// TIA Portal V17 export
// export: Created 2025-03-05T08:03:47.5129937Z, ExportSetting WithDefaults, DisplayName Totally Integrated Automation Portal, DisplayVersion V17 Update 8, DisplayName TIA Portal Openness, DisplayVersion V17 Update 8, DisplayName TIA Portal Version Control Interface, DisplayVersion V17, DisplayName SINAMICS Startdrive Advanced, DisplayVersion V17 SP2, DisplayName SINAMICS Startdrive G110M, G120, G120C, G120D, G120P, G115D, DisplayVersion V17 SP2, DisplayName SINAMICS Startdrive G130, G150, S120, S150, SINAMICS MV, S210, DisplayVersion V17 SP2, DisplayName STEP 7 Professional, DisplayVersion V17 Update 8, DisplayName SINUMERIK ONE STEP 7 Toolbox, DisplayVersion V17 Update 12, DisplayName SINUMERIK 840D sl STEP 7 Toolbox, DisplayVersion V17 Update 12, DisplayName STEP 7 Safety, DisplayVersion V17 Update 6, DisplayName WinCC Advanced, DisplayVersion V17 Update 8
TYPE "AXIS_SAFETY_IN"
// stored: IsFailsafeCompliant true
   STRUCT
      STO_Active : Bool;   // SAFE TORQUE OFF ACTIVE
      SS1_Active : Bool;   // SAFE STOP 1 ACTIVE
      SS2_Active : Bool;   // SAFE STOP 2 ACTIVE
      SOS_Active : Bool;   // SAFE OPERATING STOP ACTIVE
      SLS_Active : Bool;   // SAFE LIMITED SPEED ACTIVE
      Reserved_Input_1 : Bool;
      SLP_Active : Bool;   // SAFETY LOGIC PROGRAMME ACTIVE
      Int_Event_Active : Bool;   // INTERNAL EVENT ACTIVE
      Reserved_Input_2 : Bool;
      SLS_BIT_0_ACTIVE : Bool;   // SAFE LIMITED SPEED BIT 0 ACTIVE
      SLS_BIT_1_ACTIVE : Bool;   // SAFE LIMITED SPEED BIT 1 ACTIVE
      Reserved_Input_3 : Bool;
      SDI_POS_ACTIVE : Bool;   // SAFE DIRECTION POSITIVE ACTIVE
      SDI_NEG_ACTIVE : Bool;   // SAFE DIRECTION NEGATIVE ACTIVE
      Reserved_Input_4 : Bool;
      "SSM_n<nx" : Bool;   // SAFE SPEED MONITOR N<NX
      Reserved_Input_5 : Bool;
      Reserved_Input_6 : Bool;
      Reserved_Input_7 : Bool;
      SLP_RANGE_ACTIVE : Bool;   // SAFETY LOGIC PROGRAMME RANGE ACTIVE
      Reserved_Input_8 : Bool;
      Reserved_Input_9 : Bool;
      SAFE_POS_VALID : Bool;   // SAFE POSITION VALID
      SAFELY_REFERENCED : Bool;   // SAFELY REFERENCED
      "F-DI_0" : Bool;
      "F-DI_1" : Bool;
      "F-DI_2" : Bool;
      SS2E_ESR : Bool;   // SAFE STOP 2 EXTENDED ESR
      SS2E_ACTIVE : Bool;   // SAFE STOP 2 EXTENDED ACTIVE
      SOS_SELECTED : Bool;   // SAFE OPERATING STOP SELECTED
      SLP_UPPER_LIMIT : Bool;   // SAFETY LOGIC PROGRAMME UPPER LIMIT
      SLP_LOWER_LIMIT : Bool;   // SAFETY LOGIC PROGRAMME LOWER LIMIT
   END_STRUCT;
END_TYPE
